TYPE ST_Auto_UpperFeedInConveyorCommand EXTENDS ST_CommandBasic :
STRUCT
END_STRUCT
END_TYPE

(* stored: Version 1.1.0.1, ProductVersion 3.1.4024.13
   DUT ST_Auto_UpperFeedInConveyorCommand: Id {c6f47e0b-4c92-4e6d-adca-4eb6a117ff63} *)
